GLOBALCONSTANTS USERFUNC_e (* Global constants *)
  (* Standard: 61499-1 *)
  (* Version 1.0, 2025-09-04, franz *)
  PACKAGE isobus::pgn;
  VAR_GLOBAL CONSTANT
    working_set_master : SINT := 0;
    task_controller : SINT := 1;
    virtual_terminal : SINT := 2;
    tractor_ecu : SINT := 3;
    auxiliary : SINT := 4;
    sequence_control_master : SINT := 5;
    working_set_member : SINT := 6;
    steering_control : SINT := 7;
    off_vehicle_gateway : SINT := 8;
    network_interconnection_unit : SINT := 9;
    unknown : SINT := 10;
    file_server : SINT := 11;
    virtual_cf : SINT := 12;
    bridged_cf : SINT := 13; (* virtual CF on this network segment managed from the NIU *)
    datalogger : SINT := 14; (* NIU bridged CF on this network segment *)
    tim_server : SINT := 16;
    tim_server_slave : SINT := 17;
    sequence_control_client : SINT := 18; (* < Use only in clients see IsoClientsReadListofExtHandles() *)
    all_clients : SINT := 20;
    all_server : SINT := 21;
    undefined : SINT := -1;
  END_VAR
END_GLOBALCONSTANTS
